TYPE U_Pixel : UNION
		Pdo	   : UDINT;
		Colors : ST_Colors;
	END_UNION
END_TYPE

(* stored: Version 1.1.0.1
   DUT U_Pixel: Id {876bdec5-0fe4-4ceb-b219-b7ad99271cd2} *)
